(* PLC project  *)

CONFIGURATION Application
  RESOURCE Application ON PLC
    TASK BusTask(INTERVAL := T#10ms, PRIORITY := 11);
    PROGRAM app WITH BusTask : app;
  END_RESOURCE
END_CONFIGURATION
